TYPE "HU_Pump_HMI"
VERSION : 0.1
// Block: HU_Pump_HMI
   STRUCT
      Alarm : Bool;
      ManStart : Bool;
      PumpRunning : Bool;
      PressureRunning : Bool;
   END_STRUCT;

END_TYPE
